Yaskawa INFORM job: MAT.JBI

/JOB
//NAME MAT
//POS
///NPOS 3,0,0,0
///TOOL 0
///PULSE
C000=-4579,41009,-34828,-12396,14045,2534
C001=-32849,46293,-36172,-10262,9703,3381
C002=-27377,50757,-36172,-7742,12531,3381
//INST
///DATE 2014/10/07 18:50
///ATTR 0,0,0,0,0,0,0,0,0,0,0,0,0,0,0,0
///FRAME BASE
NOP
*1
MOVJ C000 VJ=40.00 CONT
MOVJ C001 VJ=40.00 CONT
MOVJ C002 VJ=40.00 CONT
JUMP *1
END
